GetFilter := THIS^.aiFilter[nFilterNumber];
END_METHOD

{warning 'Add method implementation '}
METHOD MoveToFilter
VAR_INPUT
    iFilter : I_HE_SATT_Filter;
    fThickness : LREAL;
END_VAR
END_METHOD


PROPERTY NumberOfSlots : INT
GET

NumberOfSlots := THIS^.nNumberOfSlots;
END_GET
SET

THIS^.nNumberOfSlots := NumberOfSlots;
END_SET
END_PROPERTY

{warning 'Add method implementation '}
METHOD RegisterFilter
VAR_INPUT
	iFilter	: I_HE_SATT_Filter;
END_VAR
END_METHOD


METHOD PUBLIC SetFilter
VAR_INPUT
	nFilterNumber : INT;
    iFilter : I_HE_SATT_Filter;
END_VAR

THIS^.aiFilter[nFilterNumber] := iFilter;
END_METHOD

{warning 'Add property implementation'}
PROPERTY Status : REFERENCE TO ST_HE_SATT_Status
GET
END_GET
END_PROPERTY

END_FUNCTION_BLOCK

// ---- Tests/Test Doubles/FB_HE_SATT_FilterHolderSelectorTestDouble.TcPOU

FUNCTION_BLOCK FB_HE_SATT_FilterHolderSelectorTestDouble IMPLEMENTS I_HE_SATT_FilterHolderSelector
VAR
    abSelectedHolder : ARRAY[1..PL_HE_SATT_Parameters.nNumHolders] OF BOOL;
END_VAR

{warning 'Add method implementation '}
METHOD CoupleHolders
VAR_INPUT
	abCoupledHolders	: ARRAY [1..PL_HE_SATT_Parameters.nNumHolders] OF BOOL;
END_VAR
END_METHOD


METHOD CouplingRulesSatisfied : BOOL
VAR_INPUT
	iFilterCombination	: I_HE_SATT_FilterCombination;
END_VAR

CouplingRulesSatisfied := TRUE;
END_METHOD


METHOD DeselectHolder
VAR_INPUT
	nHolderNumber	: INT;
END_VAR

THIS^.abSelectedHolder[nHolderNumber] := FALSE;
END_METHOD


METHOD IsSelected : BOOL
VAR_INPUT
	nHolderNumber	: INT;
END_VAR

IsSelected := THIS^.abSelectedHolder[nHolderNumber];
END_METHOD


METHOD Reset
VAR
    nIteratorHolder : INT;
END_VAR

FOR nIteratorHolder := 1 TO PL_HE_SATT_Parameters.nNumHolders BY 1 DO
    THIS^.abSelectedHolder[nIteratorHolder] := FALSE;
END_FOR
END_METHOD

{warning 'Add method implementation '}
METHOD SelectAll
END_METHOD


METHOD SelectHolder
VAR_INPUT
	nHolderNumber	: INT;
END_VAR

THIS^.abSelectedHolder[nHolderNumber] := TRUE;
END_METHOD

END_FUNCTION_BLOCK

// ---- Tests/HE_SATT/FB_HE_SATT_FilterCombinationToTransmission_Test.TcPOU

FUNCTION_BLOCK FB_HE_SATT_FilterCombinationToTransmission_Test EXTENDS FB_TestSuite


GivenCombinationExpectCorrectTransmission();


METHOD PRIVATE GivenCombinationExpectCorrectTransmission
VAR
    fbFilterHolderTestDouble : FB_HE_SATT_FilterHolderTestDouble;    

    fbFilterConstantThickness : FB_HE_SATT_FilterConstantThickness(
        iHolder := fbFilterHolderTestDouble,
        eDefaultMaterial := E_HE_SATT_FilterMaterial.Diamond,
        eDefaultStatus := E_HE_SATT_FilterStatus.ENABLED,
        fDefaultLength := 1.0,
        fDefaultThickness := 1e-3
    );
    
    fbFilterWedgeSilicon : FB_HE_SATT_FilterWedge(
        iHolder := fbFilterHolderTestDouble,
        eDefaultMaterial := E_HE_SATT_FilterMaterial.Silicon,
        eDefaultStatus := E_HE_SATT_FilterStatus.ENABLED,
        fDefaultLength := 2.0,
        fDefaultThicknessAt0 := 1e-5,
        fDefaultThicknessAtLength := 2e-5
    );
    
    fbFilterWedgeGermanium : FB_HE_SATT_FilterWedge(
        iHolder := fbFilterHolderTestDouble,
        eDefaultMaterial := E_HE_SATT_FilterMaterial.Germanium,
        eDefaultStatus := E_HE_SATT_FilterStatus.ENABLED,
        fDefaultLength := 3.0,
        fDefaultThicknessAt0 := 2e-4,
        fDefaultThicknessAtLength := 1e-4
    );
    
    fbFilterCombination : FB_HE_SATT_FilterCombination;
    
    fbScatteringFactorLookup : FB_ScatteringFactorLookupCXRO;
    
    fbFilterToTransmission : FB_HE_SATT_FilterToTransmission(
        iScatteringFactorLookup := fbScatteringFactorLookup
    );

    // Subject under test
    fbFilterCombinationToTransmission : FB_HE_SATT_FilterCombinationToTransmission(
        iFilterToTransmission := fbFilterToTransmission
    );
    
    // Variables for the test
    fMinimumTransmissionExpected : LREAL;
    fMaximumTransmissionExpected : LREAL;
    fMinimumTransmissionResult : LREAL;
    fMaximumTransmissionResult : LREAL;
    fAllowableDelta : LREAL;
END_VAR

TEST('GivenCombinationExpectCorrectTransmission');

fAllowableDelta := 1e-4;

fMinimumTransmissionExpected := 0.48445900560318955 * 0.8614762404598273 * 0.021584989971438408;
fMaximumTransmissionExpected := 0.48445900560318955 * 0.9281574437884056 * 0.14691831053833423;

fbFilterCombination.AddFilter(nHolderNumber := 1, iFilter := fbFilterConstantThickness);
fbFilterCombination.AddFilter(nHolderNumber := 3, iFilter := fbFilterWedgeSilicon);
fbFilterCombination.AddFilter(nHolderNumber := 5, iFilter := fbFilterWedgeGermanium);

fbFilterCombinationToTransmission.CalculateTransmission(
    fPhotonEnergy_eV := 10000.0,
    iFilterCombination := fbFilterCombination,
    fMinimumTransmission => fMinimumTransmissionResult,
    fMaximumTransmission => fMaximumTransmissionResult
);

AssertEquals_LREAL(
    Expected := fMinimumTransmissionExpected,
    Actual := fMinimumTransmissionResult,
    Delta := fAllowableDelta,
    Message := 'Incorrect minimum transmission computed.'
);
AssertEquals_LREAL(
    Expected := fMaximumTransmissionExpected,
    Actual := fMaximumTransmissionResult,
    Delta := fAllowableDelta,
    Message := 'Incorrect maximum transmission computed.'
);

TEST_FINISHED();
END_METHOD

END_FUNCTION_BLOCK

// ---- Tests/HE_SATT/FB_HE_SATT_FilterToTransmission_Test.TcPOU

FUNCTION_BLOCK FB_HE_SATT_FilterToTransmission_Test EXTENDS FB_TestSuite


GivenFilterExpectCorrectTransmission();


METHOD PRIVATE GivenFilterExpectCorrectTransmission
VAR
    fbFilterHolderTestDouble : FB_HE_SATT_FilterHolderTestDouble;    

    fbFilterConstantThickness : FB_HE_SATT_FilterConstantThickness(
        iHolder := fbFilterHolderTestDouble,
        eDefaultMaterial := E_HE_SATT_FilterMaterial.Diamond,
        eDefaultStatus := E_HE_SATT_FilterStatus.ENABLED,
        fDefaultLength := 1.0,
        fDefaultThickness := 1e-3
    );
    
    fbFilterWedgeSilicon : FB_HE_SATT_FilterWedge(
        iHolder := fbFilterHolderTestDouble,
        eDefaultMaterial := E_HE_SATT_FilterMaterial.Silicon,
        eDefaultStatus := E_HE_SATT_FilterStatus.ENABLED,
        fDefaultLength := 2.0,
        fDefaultThicknessAt0 := 1e-5,
        fDefaultThicknessAtLength := 2e-5
    );
    
    fbFilterWedgeGermanium : FB_HE_SATT_FilterWedge(
        iHolder := fbFilterHolderTestDouble,
        eDefaultMaterial := E_HE_SATT_FilterMaterial.Germanium,
        eDefaultStatus := E_HE_SATT_FilterStatus.ENABLED,
        fDefaultLength := 3.0,
        fDefaultThicknessAt0 := 2e-4,
        fDefaultThicknessAtLength := 1e-4
    );
    
    fbScatteringFactorLookup : FB_ScatteringFactorLookupCXRO;

    // Subject under test
    fbFilterToTransmission : FB_HE_SATT_FilterToTransmission(
        iScatteringFactorLookup := fbScatteringFactorLookup
    );
    
    // Variables for the test
    fMinimumTransmissionExpected : LREAL;
    fMaximumTransmissionExpected : LREAL;
    fMinimumTransmissionResult : LREAL;
    fMaximumTransmissionResult : LREAL;
    fAllowableDelta : LREAL;
END_VAR

TEST('GivenFilterExpectCorrectTransmission');

fAllowableDelta := 1e-4;

fMinimumTransmissionExpected := 0.4844590049714352;
fMaximumTransmissionExpected := 0.4844590049714352;

fbFilterToTransmission.CalculateTransmission(
    fPhotonEnergy_eV := 10000.0,
    iFilter := fbFilterConstantThickness,
    fMinimumTransmission => fMinimumTransmissionResult,
    fMaximumTransmission => fMaximumTransmissionResult
);

AssertEquals_LREAL(
    Expected := fMinimumTransmissionExpected,
    Actual := fMinimumTransmissionResult,
    Delta := fAllowableDelta,
    Message := 'Diamond filter with constant thickness minimum transmission was incorrect.'
);
AssertEquals_LREAL(
    Expected := fMaximumTransmissionExpected,
    Actual := fMaximumTransmissionResult,
    Delta := fAllowableDelta,
    Message := 'Diamond filter with constant thickness miaximum transmission was incorrect.'
);

fMinimumTransmissionExpected := 0.0005707894566343199;
fMaximumTransmissionExpected := 0.023891200401702714;

fbFilterToTransmission.CalculateTransmission(
    fPhotonEnergy_eV := 1000,
    iFilter := fbFilterWedgeSilicon,
    fMinimumTransmission => fMinimumTransmissionResult,
    fMaximumTransmission => fMaximumTransmissionResult
);

AssertEquals_LREAL(
    Expected := fMinimumTransmissionExpected,
    Actual := fMinimumTransmissionResult,
    Delta := fAllowableDelta,
    Message := 'Silicon filter with wedge thickness minimum transmission was incorrect.'
);
AssertEquals_LREAL(
    Expected := fMaximumTransmissionExpected,
    Actual := fMaximumTransmissionResult,
    Delta := fAllowableDelta,
    Message := 'Silicon filter with wedge thickness maximum transmission was incorrect.'
);

fMinimumTransmissionExpected := 0.010728580119616998;
fMaximumTransmissionExpected := 0.10357885942419427;

fbFilterToTransmission.CalculateTransmission(
    fPhotonEnergy_eV := 20000,
    iFilter := fbFilterWedgeGermanium,
    fMinimumTransmission => fMinimumTransmissionResult,
    fMaximumTransmission => fMaximumTransmissionResult
);

AssertEquals_LREAL(
    Expected := fMinimumTransmissionExpected,
    Actual := fMinimumTransmissionResult,
    Delta := fAllowableDelta,
    Message := 'Germanium filter with wedge thickness minimum transmission was incorrect.'
);
AssertEquals_LREAL(
    Expected := fMaximumTransmissionExpected,
    Actual := fMaximumTransmissionResult,
    Delta := fAllowableDelta,
    Message := 'Germanium filter with wedge thickness maximum transmission was incorrect.'
);

TEST_FINISHED();
END_METHOD

END_FUNCTION_BLOCK

// ---- Tests/HE_SATT/FB_HE_SATT_UserRequest_Test.TcPOU

FUNCTION_BLOCK FB_HE_SATT_UserRequest_Test EXTENDS FB_TestSuite
VAR
END_VAR


GivenApplyCommandedStartNewConfiguration();


METHOD PRIVATE GivenApplyCommandedStartNewConfiguration
VAR
    fbHE_SATT_SequenceTestDouble : FB_HE_SATT_SequenceTestDouble;
    
    // Subject under test
    fbHE_SATT_UserRequest : FB_HE_SATT_UserRequest(iHE_SATT_Sequence := fbHE_SATT_SequenceTestDouble);
END_VAR

TEST('GivenApplyCommandedStartNewConfiguration');

fbHE_SATT_UserRequest.RequestTransmission(
    fRequestedTransmission := 0.8,
    eRequestedRoundingMode := E_HE_SATT_RoundingMode.FIRST_ABOVE_WITHIN_TOLERANCE,
    fRequestedAllowableTolerance := 1e-2
);

AssertEquals_LREAL(
    Expected := 0.0,
    Actual := fbHE_SATT_SequenceTestDouble.GetStartTransmissionValue(),
    Delta := 0.0001,
    Message := 'Not correct value #1'
);

AssertEquals_UINT(
    Expected := E_HE_SATT_RoundingMode.FIRST_BELOW_WITHIN_TOLERANCE,
    Actual := fbHE_SATT_SequenceTestDouble.GetStartRoundingModeValue(),
    Message := 'Not correct value #2'
);

AssertEquals_LREAL(
    Expected := 0.0,
    Actual := fbHE_SATT_SequenceTestDouble.GetStartAllowableToleranceValue(),
    Delta := 0.0001,
    Message := 'Not correct value #3'
);

fbHE_SATT_UserRequest.ApplyConfig();

AssertEquals_LREAL(
    Expected := 0.8,
    Actual := fbHE_SATT_SequenceTestDouble.GetStartTransmissionValue(),
    Delta := 0.0001,
    Message := 'Not correct value #4'
);

AssertEquals_UINT(
    Expected := E_HE_SATT_RoundingMode.FIRST_ABOVE_WITHIN_TOLERANCE,
    Actual := fbHE_SATT_SequenceTestDouble.GetStartRoundingModeValue(),
    Message := 'Not correct value #5'
);

AssertEquals_LREAL(
    Expected := 1e-2,
    Actual := fbHE_SATT_SequenceTestDouble.GetStartAllowableToleranceValue(),
    Delta := 0.0001,
    Message := 'Not correct value #6'
);

TEST_FINISHED();
END_METHOD

END_FUNCTION_BLOCK

// ---- Tests/Test Doubles/FB_HE_SATT_SequenceTestDouble.TcPOU

FUNCTION_BLOCK FB_HE_SATT_SequenceTestDouble IMPLEMENTS I_HE_SATT_Sequence
VAR
    fStartTransmissionValue : LREAL;
    eStartRoundingModeValue : E_HE_SATT_RoundingMode;
    fStartAllowableToleranceValue : LREAL;
END_VAR


METHOD PUBLIC GetStartAllowableToleranceValue : LREAL

GetStartAllowableToleranceValue := THIS^.fStartAllowableToleranceValue;
END_METHOD


METHOD PUBLIC GetStartRoundingModeValue : E_HE_SATT_RoundingMode

GetStartRoundingModeValue := THIS^.eStartRoundingModeValue;
END_METHOD


METHOD PUBLIC GetStartTransmissionValue : LREAL

GetStartTransmissionValue := THIS^.fStartTransmissionValue;
END_METHOD


METHOD Start
VAR_INPUT
    fRequestedTransmission : LREAL; // [0.0 - 1.0]
    eRequestedRoundingMode : E_HE_SATT_RoundingMode;
    fRequestedAllowableTolerance : LREAL;
END_VAR

THIS^.fStartTransmissionValue := fRequestedTransmission;
THIS^.eStartRoundingModeValue := eRequestedRoundingMode;
THIS^.fStartAllowableToleranceValue := fRequestedAllowableTolerance;
END_METHOD

END_FUNCTION_BLOCK

// ---- Tests/PRG_TEST.TcPOU
{attribute 'analysis' := '-33'}
PROGRAM PRG_TEST
VAR
    //fbATMTest: FB_ATMTest;
    fbHE_SATT_EpicsHeartBeatTest : FB_HE_SATT_EpicsHeartBeat_Test;
    fbHE_SATT_FilterCombinationCollector_Test : FB_HE_SATT_FilterCombinationCollector_Test;
    fbHE_SATT_FilterCombinationFinder_Test : FB_HE_SATT_FilterCombinationFinder_Test;
    fbHE_SATT_FilterCombinationToTransmission_Test : FB_HE_SATT_FilterCombinationToTransmission_Test;
    fbHE_SATT_FilterHolderSelector_Test : FB_HE_SATT_FilterHolderSelector_Test;
    fbHE_SATT_FilterToTransmission_Test : FB_HE_SATT_FilterToTransmission_Test;
    fbHE_SATT_FindOptimalFilterCombination_Test : FB_HE_SATT_FindOptimalFilterCombination_Test;
    fbHE_SATT_UserRequest_Test : FB_HE_SATT_UserRequest_Test;
//     fbLICTest: FB_LICTest;
//     fbPPMTest: FB_PPMTest;
//     fbREFTest: FB_REFTest;
//     fbSATTTest: FB_SATTTest;
//     fbSlitsPowerTest: FB_SLITS_POWERTest;
//     fbWFSTest: FB_WFSTest;
//     fbXPIMTest: FB_XPIMTest;
//     fbCheckPositionStateWriteTest: FB_CheckPositionStateWriteTest;
//     fbCCTempSensorTest: FB_CC_TempSensorTest;
//
//     fbSetupJson: FB_PMPSJsonTestHelper;
//     astBeamParams: ARRAY[0..9] OF ST_DbStateParams;
//     nIter: UINT;
END_VAR


// Setup a fake db export for the test suite
// FOR nIter := 0 TO 9 DO
//     astBeamParams[nIter].stBeamParams := PMPS_GVL.cstFullBeam;
//     astBeamParams[nIter].sPmpsState := CONCAT('T', UINT_TO_STRING(nIter));
//     astBeamParams[nIter].stReactiveParams.nTempSP := nIter + 20;
// END_FOR
// fbSetupJson(
//     astBeamParams := astBeamParams,
//     bExecute := TRUE,
//     sDevNAme := 'DEVICE',
// );
// Run the tests
TcUnit.RUN();

END_PROGRAM
